Fanuc KAREL source: V_SET_REF.kl

PROGRAM T
%NOLOCKGROUP
VAR
 v0 : STRING[40]
 v1 : INTEGER
BEGIN
 V_SET_REF(v0, v1)
END T
